// TIA Portal V19 export
DATA_BLOCK "_IOL_VM_Burk_8691r3Param"   // DB502
TITLE = Valve Monitoring Params for Burkett 8691 rev.3
{ S7_Optimized_Access := 'TRUE' }
// stored: AutoNumber false, MemoryReserve 0
   VAR RETAIN
      VM_IOL_Params : "_ILO_VM_Burkett8691rev3";
   END_VAR
BEGIN
   VM_IOL_Params.StandardStructure.Parameter.ValveCyclesProgress.value := 0.0;
END_DATA_BLOCK
